# EPICS substitutions: test/iocTest/TestApp/Db/test.substitutions
file test.template {
pattern
	{ Slot_OUT_Module, Slot_INP_Module }

	{ "3", "4"}
}
